FUNCTION_BLOCK StepChainResetter IMPLEMENTS Callback
VAR_INPUT
	stepReference:REFERENCE TO UDINT;
END_VAR
VAR_OUTPUT
END_VAR
VAR
END_VAR


(* This is method get's exectued by the framework when the callback is triggered.
 It returns a step number which might be used together with Await to jump to a certain chain step
 after the callback code has been executed.*)
METHOD execute : UDINT
stepReference := 0;
END_METHOD

END_FUNCTION_BLOCK

(* stored: Version 1.1.0.1, ProductVersion 3.1.4024.12
   POU StepChainResetter: Id {dc7dbcc0-ea5e-4b09-bc26-2e6958033dce}, SpecialFunc None
   Method execute: Id {9c3e1ca9-c3f1-4fcb-a1dc-e54cf5122f74} *)
